# EPICS substitutions: db/SmarAct/ecmcMCS2.substitutions
file "ecmcEcSlave.template"
{
  pattern {}
          {}
}

file "ecmcMCS_generic.template"
{
  pattern {}
          {}
}

file "ecmcDS402_Drive_CSP.template"
{
  pattern {CH_ID, LINR,    ESLO,   EOFF,   EGU,        PREC, LOW, LOLO, HIGH, HIHI, HYST, LLSV,       LSV,        HSV,        HHSV      }
          {01,     "SLOPE", 1,      0,      "Raw",      0,    0,   0,    0,    0,    0,    "NO_ALARM", "NO_ALARM", "NO_ALARM", "NO_ALARM"}
          {02,     "SLOPE", 1,      0,      "Raw",      0,    0,   0,    0,    0,    0,    "NO_ALARM", "NO_ALARM", "NO_ALARM", "NO_ALARM"}
          {03,     "SLOPE", 1,      0,      "Raw",      0,    0,   0,    0,    0,    0,    "NO_ALARM", "NO_ALARM", "NO_ALARM", "NO_ALARM"}
}

file "ecmcEncoder_32bit.template"
{
  pattern {CH_ID, LINR,    ESLO,   EOFF,   EGU,        PREC, LOW, LOLO, HIGH, HIHI, HYST, LLSV,       LSV,        HSV,        HHSV      }
          {01,     "SLOPE", 1,      0,      "Raw",      0,    0,   0,    0,    0,    0,    "NO_ALARM", "NO_ALARM", "NO_ALARM", "NO_ALARM"}
          {02,     "SLOPE", 1,      0,      "Raw",      0,    0,   0,    0,    0,    0,    "NO_ALARM", "NO_ALARM", "NO_ALARM", "NO_ALARM"}
          {03,     "SLOPE", 1,      0,      "Raw",      0,    0,   0,    0,    0,    0,    "NO_ALARM", "NO_ALARM", "NO_ALARM", "NO_ALARM"}
}

file "ecmcMCS2_custom.template"
{
  pattern {CH_ID}
          {01   }
          {02   }
          {03   }
}

# ecmcDS402Enable
file "ecmcDS402Enable-chX.template"
{
  pattern {CH_ID}
          {01   }
          {02   }
          {03   }
}
